// TwinCAT 3 PLC project PLCStudent
// ProgramVersion: 3.1.4026.21
// libraries:
//   Tc2_Standard, * (Beckhoff Automation GmbH)
//   Tc2_System, * (Beckhoff Automation GmbH)
//   Tc3_Module, * (Beckhoff Automation GmbH)
//   VisuSymbols, 4.5.0.0 (System)
// project tree:
//   / GlobalTextList.TcGTLO, PlcTask.TcTTO, Visualization Manager.TcVMO (not stored)
//   GVLs/ GVL.TcGVL (not stored), GVL_CTRL.TcGVL (not stored)
//   POUs/ FB_AGVComm.TcPOU (not stored), MAIN.TcPOU, RunStudent.TcPOU (not stored)
//   VISUs/ Visualization.TcVIS
// (motion and I/O tree: see PLC project plcsim)
// real-time tasks:
//   TASK PlcTask: cycle T#20ms, priority 20, ADS port 350
// variable links:
//   PLCSim/PLCSim Instance <-> PLCStudent/PLCStudent Instance
//     PlcTask Inputs/GVL.iiGotoPos <-> PlcTask Outputs/GVL.iiGotoPos
//     PlcTask Inputs/GVL.ixPLCStrobe <-> PlcTask Outputs/GVL.ixPLCStrobe
//     PlcTask Outputs/GVL.qiAtPos <-> PlcTask Inputs/GVL.iiAtPos
//     PlcTask Outputs/GVL.qxAGVStrobe <-> PlcTask Inputs/GVL.ixAGVStrobe

CONFIGURATION PLCStudent
    RESOURCE PLC ON TwinCAT3
        TASK PlcTask(INTERVAL := T#20ms, PRIORITY := 20);
        PROGRAM MAIN WITH PlcTask : MAIN;
    END_RESOURCE
END_CONFIGURATION

// ---- POUs/MAIN.TcPOU
PROGRAM MAIN
VAR
    
END_VAR

RunStudent();

END_PROGRAM

// ---- GlobalTextList.TcGTLO
TEXTLIST GlobalTextList
  791 = 'GVL.iiAtPos'
  94 = 'hhh'
  315 = 'Moving'
  952 = 'Position = %s'
  214 = 'Ready'
  823 = 'Reset'
  221 = 'START'
  785 = 'Start'
  886 = 'Stop'
  523 = 'Target selection\n1 = HOME\n2 = A\n3 = B\n4 = C\n5 = D'
END_TEXTLIST

// ---- VISUs/Visualization.TcVIS
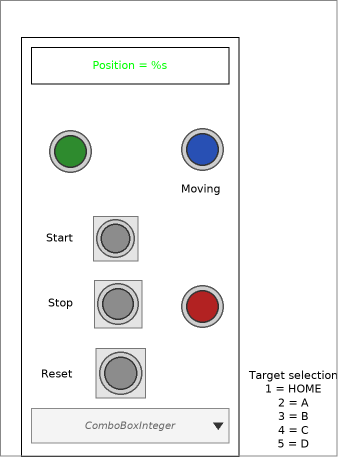
VISUALIZATION Visualization  // 338x457
    Rectangle (21,37 218x420)
    PushSwitch (93,280 50x48), variable: GVL_CTRL.xStopPB, behaviour: TAP, style: Switch-PushSwitch-Gray
    PushSwitch (93,348 55x50), variable: GVL_CTRL.xResetPB, behaviour: TAP, style: Switch-PushSwitch-Gray
    Label (31,359 52x30), "Reset"
    Label (38,288 45x30), "Stop"
    PushSwitch (93,214 45x49), variable: GVL_CTRL.xStartPB, behaviour: TAP, style: Switch-PushSwitch-Gray
    Label (31,223 57x30), "Start"
    Lamp1 (46,120 49x63), variable: GVL_CTRL.xReadyLamp, style: Lamp-Lamp1-Green
    Lamp1 (178,120 49x59), variable: GVL_CTRL.xMovingLamp, style: Lamp-Lamp1-Blue
    Label (126,174 150x30), "Moving"
    Lamp1 (178,280 49x53), variable: GVL_CTRL.xStopLamp, style: Lamp-Lamp1-Red
    Rectangle (31,47 198x37), "Position = %s", text variable: GVL.iiAtPos
    ComboBoxInteger (31,408 198x35), variable: GVL_CTRL.iTarget
    Label (249,362 89x95), "Target selection 1 = HOME 2 = A 3 = B 4 = C 5 = D"
END_VISUALIZATION
